Staubli VAL3: setPalletPos.pgx

public program setPalletPos(string x_sItem, num x_nValue)
  local num i
  local string l_sName
  local num l_nPos
begin
  // scan it
  if isDefined(pt:tTraj[x_sItem])
    // redefine the position
    pt:tTraj[x_sItem].nIndex=x_nValue
  endIf
end
